TYPE (* Write register communication *)
  (* Description: Copyright (c) 2026 Monika Wenger This program and the accompanying materials are made available under the terms of the Eclipse Public License 2.0 which is available at https://www.eclipse.org/legal/epl-2.0/ SPDX-License-Identifier: EPL-2.0 *)
  (* Version 3.0, 2026-07-21, Monika Wenger *)
  PACKAGE eclipse4diac::io::wago;
  RegComCmd : STRUCT
    RegNr : USINT;
    REG_D0 : BYTE;
    REG_D1 : BYTE;
  END_STRUCT;
END_TYPE
